(* IEC 61131-3 sources: Word/plc-course/03-data-types-and-addressing/labs/starter, 3 files *)

(* ---- 03-1-status-and-command-words.st ---- *)
(* Lab 03-1: Status word and command word - packing BOOLs into a WORD and back.
   Module 03 (Numbers, data types and addressing). STARTER - the declarations are done for you;
   write the logic where it says TODO, then run:
     python3 tools/plctest.py 03-data-types-and-addressing/labs/starter/03-1-status-and-command-words.st

   A pump station PLC exchanges data with SCADA through two 16-bit registers:
     StatusWord (PLC -> SCADA): bit n = status flag n (bits 0..7), bit 15 = command word rejected
     CmdWord    (SCADA -> PLC): bits 0..7 = eight commands, bits 8..15 reserved (must be 0)
   MATIEC has no bit access such as CmdWord.3, so use shifts and masks (see the README). CODESYS
   (CmdWord.3), TIA Portal (CmdWord.%X3) and Logix (MyDint.3) let you address bits directly. *)

PROGRAM PumpWords
  VAR (* I/O: eight status inputs = one byte of a digital input card (%IB0) *)
    Running       AT %IX0.0 : BOOL;  (* bit 0: pump running (contactor auxiliary contact) *)
    InAuto        AT %IX0.1 : BOOL;  (* bit 1: Hand-Off-Auto selector in AUTO *)
    Tripped       AT %IX0.2 : BOOL;  (* bit 2: motor protection relay tripped *)
    SuctionLow    AT %IX0.3 : BOOL;  (* bit 3: suction pressure low *)
    DischargeHigh AT %IX0.4 : BOOL;  (* bit 4: discharge pressure high *)
    SealLeak      AT %IX0.5 : BOOL;  (* bit 5: mechanical seal leak detected *)
    SumpHigh      AT %IX0.6 : BOOL;  (* bit 6: sump level high *)
    PanelDoorOpen AT %IX0.7 : BOOL;  (* bit 7: control panel door open *)
  END_VAR
  VAR (* SCADA interface: OpenPLC serves %MW0 and %MW1 as Modbus holding registers 1024 and 1025 *)
    StatusWord AT %MW0 : WORD;  (* PLC -> SCADA *)
    CmdWord    AT %MW1 : WORD;  (* SCADA -> PLC *)
  END_VAR
  VAR (* unpacked commands, used by the rest of the program *)
    CmdStart    : BOOL;  (* bit 0 *)
    CmdStop     : BOOL;  (* bit 1 *)
    CmdReset    : BOOL;  (* bit 2 *)
    CmdAuto     : BOOL;  (* bit 3 *)
    CmdManual   : BOOL;  (* bit 4 *)
    CmdInhibit  : BOOL;  (* bit 5 *)
    CmdLampTest : BOOL;  (* bit 6 *)
    CmdSilence  : BOOL;  (* bit 7: silence the horn *)
    CmdRejected : BOOL;  (* TRUE while a reserved bit (8..15) of CmdWord is set *)
  END_VAR

  (* TODO Part A: build StatusWord from the eight status flags (bit n = flag n)
     and set bit 15 while CmdRejected is TRUE. Bits 8..14 are always 0.
     TODO Part B: set CmdRejected when any of bits 8..15 of CmdWord is set, and
     unpack bits 0..7 of CmdWord into CmdStart..CmdSilence (all FALSE when rejected).
     Replace these placeholder lines with your logic. *)
  StatusWord := 16#0000;
  CmdStart := FALSE;
  CmdStop := FALSE;
  CmdReset := FALSE;
  CmdAuto := FALSE;
  CmdManual := FALSE;
  CmdInhibit := FALSE;
  CmdLampTest := FALSE;
  CmdSilence := FALSE;
  CmdRejected := FALSE;
END_PROGRAM

CONFIGURATION Config0
  RESOURCE Res0 ON PLC
    TASK MainTask(INTERVAL := T#10ms, PRIORITY := 0);
    PROGRAM Inst0 WITH MainTask : PumpWords;
  END_RESOURCE
END_CONFIGURATION

(* ---- 03-2-bcd-display-and-thumbwheel.st ---- *)
(* Lab 03-2: BCD display and thumbwheel - converting between binary INT and 4-digit BCD.
   Module 03 (Numbers, data types and addressing). STARTER - the declarations are done for you;
   write the logic where it says TODO, then run:
     python3 tools/plctest.py 03-data-types-and-addressing/labs/starter/03-2-bcd-display-and-thumbwheel.st

   An older batching skid has a 4-digit BCD display (16 digital outputs) and a 4-decade BCD
   thumbwheel switch (16 digital inputs). Each decimal digit uses one nibble (4 bits):
     bits 15..12 = thousands, 11..8 = hundreds, 7..4 = tens, 3..0 = units.
   So 1234 is sent as 16#1234, not as the binary value 16#04D2.
   Work out the digits yourself with / MOD SHL SHR AND OR. (MATIEC also offers
   UINT_TO_BCD_WORD and WORD_BCD_TO_UINT, but you still need your own range and
   validity checks, so try it by hand first.) *)

PROGRAM BcdPanel
  VAR (* I/O *)
    ThumbwheelBCD    AT %IW0   : WORD;  (* 16 inputs from the thumbwheel switch, 4 BCD digits *)
    DisplayBCD       AT %QW0   : WORD;  (* 16 outputs to the display, 4 BCD digits *)
    DisplayOverRange AT %QX0.0 : BOOL;  (* lamp: DisplayValue cannot be shown in 4 digits *)
    ThumbwheelFault  AT %QX0.1 : BOOL;  (* lamp: the thumbwheel reading has an invalid digit *)
  END_VAR
  VAR (* interface to the rest of the program *)
    DisplayValue : INT;  (* value to show on the display, written by other logic *)
    BatchSize    : INT;  (* decoded thumbwheel setting, 0..9999 *)
  END_VAR
  VAR (* internal: add any helper variables you need here *)
    ShowValue : INT;     (* suggestion: DisplayValue after clamping to 0..9999 *)
  END_VAR

  (* TODO Part A: clamp DisplayValue to 0..9999 (DisplayOverRange TRUE when it had to be
     clamped) and write it to DisplayBCD as four BCD digits.
     TODO Part B: decode ThumbwheelBCD into BatchSize. If any digit is 10..15, set
     ThumbwheelFault and keep the last good BatchSize.
     Replace these placeholder lines with your logic. *)
  DisplayBCD := 16#0000;
  DisplayOverRange := FALSE;
  BatchSize := 0;
  ThumbwheelFault := FALSE;
END_PROGRAM

CONFIGURATION Config0
  RESOURCE Res0 ON PLC
    TASK MainTask(INTERVAL := T#10ms, PRIORITY := 0);
    PROGRAM Inst0 WITH MainTask : BcdPanel;
  END_RESOURCE
END_CONFIGURATION

(* ---- 03-3-temperature-tenths.st ---- *)
(* Lab 03-3: Temperature in tenths - integer versus REAL arithmetic.
   Module 03 (Numbers, data types and addressing). STARTER - the declarations are done for you;
   write the logic where it says TODO, then run:
     python3 tools/plctest.py 03-data-types-and-addressing/labs/starter/03-3-temperature-tenths.st

   A temperature transmitter sends its reading as an INT in tenths of a degree Celsius
   (235 means 23.5 degC), a very common convention on Modbus devices. The program makes
     TempC      REAL degC for the HMI
     TempF      REAL degF for the HMI
     TempF_x10  INT tenths of degF, rounded to the nearest tenth, for a legacy SCADA register
   and flags readings outside the sensor's measuring range. *)

PROGRAM TempTenths
  VAR (* I/O *)
    RawTenths   AT %IW0   : INT;   (* from the transmitter: tenths of degC *)
    TempF_x10   AT %QW0   : INT;   (* to legacy SCADA: tenths of degF (Modbus holding register 0 in OpenPLC) *)
    SensorFault AT %QX0.0 : BOOL;  (* reading outside -200.0 .. +850.0 degC *)
  END_VAR
  VAR (* HMI values *)
    TempC : REAL;                  (* degC *)
    TempF : REAL;                  (* degF *)
  END_VAR
  VAR CONSTANT
    RAW_MIN : INT := -2000;        (* -200.0 degC: bottom of the Pt100 range *)
    RAW_MAX : INT := 8500;         (* +850.0 degC: top of the Pt100 range *)
  END_VAR

  (* TODO: set SensorFault when RawTenths is outside RAW_MIN..RAW_MAX.
     TODO: for good readings, calculate TempC, TempF and TempF_x10 (tenths of degF,
     rounded to the nearest tenth, correct over the whole range). On a fault, keep the
     last good values. Watch out for integer division and INT overflow.
     Replace these placeholder lines with your logic. *)
  SensorFault := FALSE;
  TempC := 0.0;
  TempF := 0.0;
  TempF_x10 := 0;
END_PROGRAM

CONFIGURATION Config0
  RESOURCE Res0 ON PLC
    TASK MainTask(INTERVAL := T#10ms, PRIORITY := 0);
    PROGRAM Inst0 WITH MainTask : TempTenths;
  END_RESOURCE
END_CONFIGURATION
